{attribute 'pack_mode' := '1'} 
TYPE ST_Beckhoff_4AI :
STRUCT
	nStatus1	AT %Q* : UINT;
	nValue1		AT %Q* : INT;
	nStatus2	AT %Q* : UINT;
	nValue2		AT %Q* : INT;
END_STRUCT
END_TYPE

(* stored: Version 1.1.0.1, ProductVersion 3.1.4024.12
   DUT ST_Beckhoff_4AI: Id {06dbb9a8-7496-038a-250a-0947d319e129} *)
